{attribute 'qualified_only'}
VAR_GLOBAL
    // Status
    {attribute 'OPC.UA.DA' := '1'}
    {attribute 'OPC.UA.DA.StructuredType' := '1'}
    g_stProcessDiagnosticsStatus : ST_ProcessDiagnosticsStatus;
END_VAR

(* stored: Version 1.1.0.1, ProductVersion 3.1.4024.16
   GVL GVL_ProcessDiagnostics: Id {4a5acf40-75b3-48cd-9044-ef8311dc738a} *)
